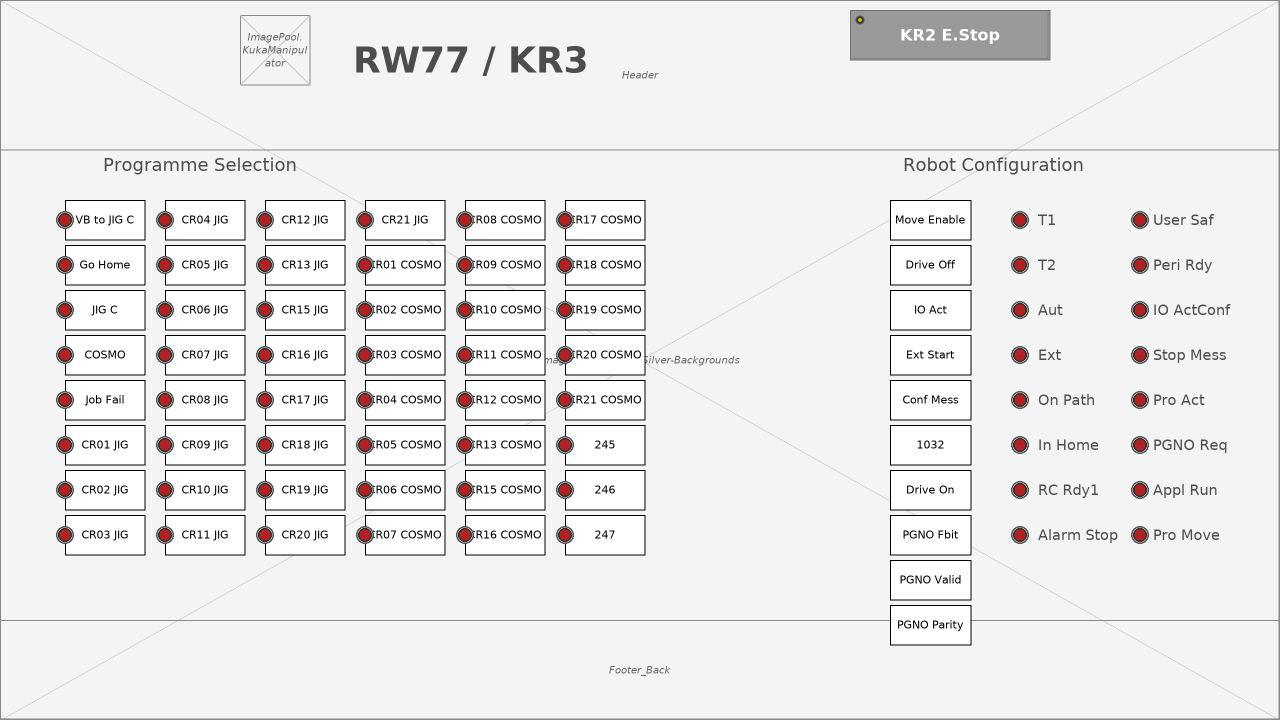
VISUALIZATION PAGE_KR2  // 1280x720
    Image (0,0 1280x720), image: ImagePool.The-New-Silver-Backgrounds
    Frame (0,620 1280x100)
        shows Footer_Back()
    Frame (0,0 1280x150)
        shows Header()
    Label (350,40 300x40), "RW77 / KR3"
    Label (100,150 250x30), "Programme Selection"
    Group (850,10 200x50)
        Button (0,0 200x50), "KR2 E.Stop"
            toggle KR2.KR2_Estop
        Lamp1 (5,5 10x10), variable: KR2.KR2_Estop, style: Lamp-Lamp1-Yellow
    Image (240,15 70x70), image: ImagePool.KukaManipulator
    Label (900,150 200x30), "Robot Configuration"
    RoundedRectangle (890,200 81x40), "Move Enable"
        toggle KR2.bOutBit[1,0]
    RoundedRectangle (890,245 81x40), "Drive Off"
        toggle KR2.bOutBit[1,1]
    RoundedRectangle (890,290 81x40), "IO Act"
        toggle KR2.bOutBit[1,2]
    RoundedRectangle (890,335 81x40), "Ext Start"
        toggle KR2.bOutBit[1,3]
    RoundedRectangle (890,380 81x40), "Conf Mess"
        toggle KR2.bOutBit[1,4]
    RoundedRectangle (890,425 81x40), "1032"
        toggle KR2.bOutBit[1,5]
    RoundedRectangle (890,470 81x40), "Drive On"
        toggle KR2.bOutBit[1,6]
    RoundedRectangle (890,515 81x40), "PGNO Fbit"
        toggle KR2.bOutBit[1,7]
    RoundedRectangle (890,560 81x40), "PGNO Valid"
        toggle KR2.bOutBit[2,0]
    RoundedRectangle (890,605 81x40), "PGNO Parity"
        toggle KR2.bOutBit[2,1]
    Label (1150,205 110x30), "User Saf"
    Label (1150,250 110x30), "Peri Rdy"
    Label (1150,295 110x30), "IO ActConf"
    Label (1150,340 110x30), "Stop Mess"
    Label (1150,385 110x30), "Pro Act"
    Label (1150,430 110x30), "PGNO Req"
    Label (1150,475 110x30), "Appl Run"
    Label (1150,520 110x30), "Pro Move"
    Label (1035,205 105x30), "T1"
    Label (1035,250 105x30), "T2"
    Label (1035,295 105x30), "Aut"
    Label (1035,340 105x30), "Ext"
    Label (1035,385 105x30), "On Path"
    Label (1035,430 105x30), "In Home"
    Label (1035,475 105x30), "RC Rdy1"
    Label (1035,520 105x30), "Alarm Stop"
    Lamp1 (1010,210 20x20), variable: KR2.bInBit[1,0], style: Lamp-Lamp1-Red
    Lamp1 (1010,255 20x20), variable: KR2.bInBit[1,1], style: Lamp-Lamp1-Red
    Lamp1 (1010,300 20x20), variable: KR2.bInBit[1,2], style: Lamp-Lamp1-Red
    Lamp1 (1010,345 20x20), variable: KR2.bInBit[1,3], style: Lamp-Lamp1-Red
    Lamp1 (1010,390 20x20), variable: KR2.bInBit[1,4], style: Lamp-Lamp1-Red
    Lamp1 (1010,435 20x20), variable: KR2.bInBit[1,5], style: Lamp-Lamp1-Red
    Lamp1 (1010,480 20x20), variable: KR2.bInBit[1,6], style: Lamp-Lamp1-Red
    Lamp1 (1010,525 20x20), variable: KR2.bInBit[1,7], style: Lamp-Lamp1-Red
    Lamp1 (1130,210 20x20), variable: KR2.bInBit[2,0], style: Lamp-Lamp1-Red
    Lamp1 (1130,255 20x20), variable: KR2.bInBit[2,1], style: Lamp-Lamp1-Red
    Lamp1 (1130,300 20x20), variable: KR2.bInBit[2,2], style: Lamp-Lamp1-Red
    Lamp1 (1130,345 20x20), variable: KR2.bInBit[2,3], style: Lamp-Lamp1-Red
    Lamp1 (1130,390 20x20), variable: KR2.bInBit[2,4], style: Lamp-Lamp1-Red
    Lamp1 (1130,435 20x20), variable: KR2.bInBit[2,5], style: Lamp-Lamp1-Red
    Lamp1 (1130,480 20x20), variable: KR2.bInBit[2,6], style: Lamp-Lamp1-Red
    Lamp1 (1130,525 20x20), variable: KR2.bInBit[2,7], style: Lamp-Lamp1-Red
    RoundedRectangle (65,200 80x40), "VB to JIG C"
        toggle KR2.bOutBit[3,0]
    RoundedRectangle (65,245 80x40), "Go Home"
        toggle KR2.bOutBit[3,1]
    RoundedRectangle (65,290 80x40), "JIG C"
        toggle KR2.bOutBit[3,2]
    RoundedRectangle (65,335 80x40), "COSMO"
        toggle KR2.bOutBit[3,3]
    RoundedRectangle (65,380 80x40), "Job Fail"
        toggle KR2.bOutBit[3,4]
    RoundedRectangle (65,425 80x40), "CR01 JIG"
        toggle KR2.bOutBit[3,5]
    RoundedRectangle (65,470 80x40), "CR02 JIG"
        toggle KR2.bOutBit[3,6]
    RoundedRectangle (65,515 80x40), "CR03 JIG"
        toggle KR2.bOutBit[3,7]
    Lamp1 (55,210 20x20), variable: KR2.bInBit[3,0], style: Lamp-Lamp1-Red
    Lamp1 (55,255 20x20), variable: KR2.bInBit[3,1], style: Lamp-Lamp1-Red
    Lamp1 (55,300 20x20), variable: KR2.bInBit[3,2], style: Lamp-Lamp1-Red
    Lamp1 (55,345 20x20), variable: KR2.bInBit[3,3], style: Lamp-Lamp1-Red
    Lamp1 (55,390 20x20), variable: KR2.bInBit[3,4], style: Lamp-Lamp1-Red
    Lamp1 (55,435 20x20), variable: KR2.bInBit[3,5], style: Lamp-Lamp1-Red
    Lamp1 (55,480 20x20), variable: KR2.bInBit[3,6], style: Lamp-Lamp1-Red
    Lamp1 (55,525 20x20), variable: KR2.bInBit[3,7], style: Lamp-Lamp1-Red
    RoundedRectangle (265,200 80x40), "CR12 JIG"
        toggle KR2.bOutBit[5,0]
    RoundedRectangle (265,245 80x40), "CR13 JIG"
        toggle KR2.bOutBit[5,1]
    RoundedRectangle (265,290 80x40), "CR15 JIG"
        toggle KR2.bOutBit[5,2]
    RoundedRectangle (265,335 80x40), "CR16 JIG"
        toggle KR2.bOutBit[5,3]
    RoundedRectangle (265,380 80x40), "CR17 JIG"
        toggle KR2.bOutBit[5,4]
    RoundedRectangle (265,425 80x40), "CR18 JIG"
        toggle KR2.bOutBit[5,5]
    RoundedRectangle (265,470 80x40), "CR19 JIG"
        toggle KR2.bOutBit[5,6]
    RoundedRectangle (265,515 80x40), "CR20 JIG"
        toggle KR2.bOutBit[5,7]
    Lamp1 (255,210 20x20), variable: KR2.bInBit[5,0], style: Lamp-Lamp1-Red
    Lamp1 (255,255 20x20), variable: KR2.bInBit[5,1], style: Lamp-Lamp1-Red
    Lamp1 (255,300 20x20), variable: KR2.bInBit[5,2], style: Lamp-Lamp1-Red
    Lamp1 (255,345 20x20), variable: KR2.bInBit[5,3], style: Lamp-Lamp1-Red
    Lamp1 (255,390 20x20), variable: KR2.bInBit[5,4], style: Lamp-Lamp1-Red
    Lamp1 (255,435 20x20), variable: KR2.bInBit[5,5], style: Lamp-Lamp1-Red
    Lamp1 (255,480 20x20), variable: KR2.bInBit[5,6], style: Lamp-Lamp1-Red
    Lamp1 (255,525 20x20), variable: KR2.bInBit[5,7], style: Lamp-Lamp1-Red
    RoundedRectangle (365,200 80x40), "CR21 JIG"
        toggle KR2.bOutBit[6,0]
    RoundedRectangle (365,245 80x40), "CR01 COSMO"
        toggle KR2.bOutBit[6,1]
    RoundedRectangle (365,290 80x40), "CR02 COSMO"
        toggle KR2.bOutBit[6,2]
    RoundedRectangle (365,335 80x40), "CR03 COSMO"
        toggle KR2.bOutBit[6,3]
    RoundedRectangle (365,380 80x40), "CR04 COSMO"
        toggle KR2.bOutBit[6,4]
    RoundedRectangle (365,425 80x40), "CR05 COSMO"
        toggle KR2.bOutBit[6,5]
    RoundedRectangle (365,470 80x40), "CR06 COSMO"
        toggle KR2.bOutBit[6,6]
    RoundedRectangle (365,515 80x40), "CR07 COSMO"
        toggle KR2.bOutBit[6,7] p2164770859=TRUE
    Lamp1 (355,210 20x20), variable: KR2.bInBit[6,0], style: Lamp-Lamp1-Red
    Lamp1 (355,255 20x20), variable: KR2.bInBit[6,1], style: Lamp-Lamp1-Red
    Lamp1 (355,300 20x20), variable: KR2.bInBit[6,2], style: Lamp-Lamp1-Red
    Lamp1 (355,345 20x20), variable: KR2.bInBit[6,3], style: Lamp-Lamp1-Red
    Lamp1 (355,390 20x20), variable: KR2.bInBit[6,4], style: Lamp-Lamp1-Red
    Lamp1 (355,435 20x20), variable: KR2.bInBit[6,5], style: Lamp-Lamp1-Red
    Lamp1 (355,480 20x20), variable: KR2.bInBit[6,6], style: Lamp-Lamp1-Red
    Lamp1 (355,525 20x20), variable: KR2.bInBit[6,7], style: Lamp-Lamp1-Red
    RoundedRectangle (465,200 80x40), "CR08 COSMO"
        toggle KR2.bOutBit[7,0]
    RoundedRectangle (465,245 80x40), "CR09 COSMO"
        toggle KR2.bOutBit[7,1]
    RoundedRectangle (465,290 80x40), "CR10 COSMO"
        toggle KR2.bOutBit[7,2]
    RoundedRectangle (465,335 80x40), "CR11 COSMO"
        toggle KR2.bOutBit[7,3]
    RoundedRectangle (465,380 80x40), "CR12 COSMO"
        toggle KR2.bOutBit[7,4]
    RoundedRectangle (465,425 80x40), "CR13 COSMO"
        toggle KR2.bOutBit[7,5]
    RoundedRectangle (465,470 80x40), "CR15 COSMO"
        toggle KR2.bOutBit[7,6]
    RoundedRectangle (465,515 80x40), "CR16 COSMO"
        toggle KR2.bOutBit[7,7] p2164770859=TRUE
    Lamp1 (455,210 20x20), variable: KR2.bInBit[7,0], style: Lamp-Lamp1-Red
    Lamp1 (455,255 20x20), variable: KR2.bInBit[7,1], style: Lamp-Lamp1-Red
    Lamp1 (455,300 20x20), variable: KR2.bInBit[7,2], style: Lamp-Lamp1-Red
    Lamp1 (455,345 20x20), variable: KR2.bInBit[7,3], style: Lamp-Lamp1-Red
    Lamp1 (455,390 20x20), variable: KR2.bInBit[7,4], style: Lamp-Lamp1-Red
    Lamp1 (455,435 20x20), variable: KR2.bInBit[7,5], style: Lamp-Lamp1-Red
    Lamp1 (455,480 20x20), variable: KR2.bInBit[7,6], style: Lamp-Lamp1-Red
    Lamp1 (455,525 20x20), variable: KR2.bInBit[7,7], style: Lamp-Lamp1-Red
    RoundedRectangle (565,200 80x40), "CR17 COSMO"
        toggle KR2.bOutBit[8,0]
    RoundedRectangle (565,245 80x40), "CR18 COSMO"
        toggle KR2.bOutBit[8,1]
    RoundedRectangle (565,290 80x40), "CR19 COSMO"
        toggle KR2.bOutBit[8,2]
    RoundedRectangle (565,335 80x40), "CR20 COSMO"
        toggle KR2.bOutBit[8,3]
    RoundedRectangle (565,380 80x40), "CR21 COSMO"
        toggle KR2.bOutBit[8,4]
    RoundedRectangle (565,425 80x40), "245"
        toggle KR2.bOutBit[8,5]
    RoundedRectangle (565,470 80x40), "246"
        toggle KR2.bOutBit[8,6]
    RoundedRectangle (565,515 80x40), "247"
        toggle KR2.bOutBit[8,7] p2164770859=TRUE
    Lamp1 (555,210 20x20), variable: KR2.bInBit[8,0], style: Lamp-Lamp1-Red
    Lamp1 (555,255 20x20), variable: KR2.bInBit[8,1], style: Lamp-Lamp1-Red
    Lamp1 (555,300 20x20), variable: KR2.bInBit[8,2], style: Lamp-Lamp1-Red
    Lamp1 (555,345 20x20), variable: KR2.bInBit[8,3], style: Lamp-Lamp1-Red
    Lamp1 (555,390 20x20), variable: KR2.bInBit[8,4], style: Lamp-Lamp1-Red
    Lamp1 (555,435 20x20), variable: KR2.bInBit[8,5], style: Lamp-Lamp1-Red
    Lamp1 (555,480 20x20), variable: KR2.bInBit[8,6], style: Lamp-Lamp1-Red
    Lamp1 (555,525 20x20), variable: KR2.bInBit[8,7], style: Lamp-Lamp1-Red
    RoundedRectangle (165,200 80x40), "CR04 JIG"
        toggle KR2.bOutBit[4,0]
    RoundedRectangle (165,245 80x40), "CR05 JIG"
        toggle KR2.bOutBit[4,1]
    RoundedRectangle (165,290 80x40), "CR06 JIG"
        toggle KR2.bOutBit[4,2]
    RoundedRectangle (165,335 80x40), "CR07 JIG"
        toggle KR2.bOutBit[4,3]
    RoundedRectangle (165,380 80x40), "CR08 JIG"
        toggle KR2.bOutBit[4,4]
    RoundedRectangle (165,425 80x40), "CR09 JIG"
        toggle KR2.bOutBit[4,5]
    RoundedRectangle (165,470 80x40), "CR10 JIG"
        toggle KR2.bOutBit[4,6]
    RoundedRectangle (165,515 80x40), "CR11 JIG"
        toggle KR2.bOutBit[4,7]
    Lamp1 (155,210 20x20), variable: KR2.bInBit[4,0], style: Lamp-Lamp1-Red
    Lamp1 (155,255 20x20), variable: KR2.bInBit[4,1], style: Lamp-Lamp1-Red
    Lamp1 (155,300 20x20), variable: KR2.bInBit[4,2], style: Lamp-Lamp1-Red
    Lamp1 (155,345 20x20), variable: KR2.bInBit[4,3], style: Lamp-Lamp1-Red
    Lamp1 (155,390 20x20), variable: KR2.bInBit[4,4], style: Lamp-Lamp1-Red
    Lamp1 (155,435 20x20), variable: KR2.bInBit[4,5], style: Lamp-Lamp1-Red
    Lamp1 (155,480 20x20), variable: KR2.bInBit[4,6], style: Lamp-Lamp1-Red
    Lamp1 (155,525 20x20), variable: KR2.bInBit[4,7], style: Lamp-Lamp1-Red
END_VISUALIZATION

(* stored: Version 1.1.0.1, ProductVersion 3.1.4024.12
   Visu PAGE_KR2: Id {aa69577d-d07a-413d-be6b-39d4cd7d2d93} *)
